# EPICS substitutions: Epics_Installation/gpib_test/gpib_test/db/Keithley2000.substitutions
file "db/keithleyHHL.db" {
    { user = "pi" }
}
